FUNCTION_BLOCK Simple (* A simple FB with a single algorithm and REQ/CNF pair *)
  (* Standard: 61499-1 *)
  (* Version 0.0, 2006-09-03, JHC, Holobloc Inc *)
  (* Compiler header: package fb.rt.template; *)
  (* Compiler classdef: SimpleFB *)
  (* Compiler Java Sun JDK 1.5.0 *)
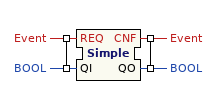
  EVENT_INPUT
    REQ WITH QI; (* Normal Execution Request *)
  END_EVENT
  EVENT_OUTPUT
    CNF WITH QO; (* Execution Confirmation *)
  END_EVENT
  VAR_INPUT
    QI : BOOL; (* Input event qualifier *)
  END_VAR
  VAR_OUTPUT
    QO : BOOL; (* Output event qualifier *)
  END_VAR
  ALGORITHM REQ IN ST: (* Normally executed algorithm *)
QO := QI;
  END_ALGORITHM
END_FUNCTION_BLOCK
